FUNCTION_BLOCK GT_DWORD (* IEC 61131-3,Table 28#5 *)
  (* Standard: 61131-3 *)
  (* Version 0.0, 2004-12-15, JHC, Rockwell Automation, Converted from SRC format. *)
  (* Compiler header: package fb.rt.plc.comp; *)
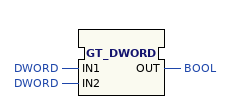
  VAR_INPUT
    IN1 : DWORD;
    IN2 : DWORD;
  END_VAR
  VAR_OUTPUT
    OUT : BOOL;
  END_VAR
END_FUNCTION_BLOCK
